Staubli VAL3: listupdate.pgx

public program listupdate(num pFirst (dimensions=1))
  local num lI
  local num lLen
  local string lStr
  local string lStr2
  local num lValue
  local num lView
  local num lX
  local num lY
  local num l_nSize
  local bool l_bEmpty
begin
  //
  // insert into the box all the data
  //
  // to prevent a negative value
  if pFirst>=0
    nFirst=pFirst
  else
    nFirst=0
  endIf
  // save the coordinate
  lValue=nBottomY-1
  // check the overFlow
  l_nSize=size(sItems)-1
  if (nFirst+nView>l_nSize)
    // reset the value
    nFirst=nView=0
  endIf
  lI=0
  // check the unKnow poblem
  if l_nSize<lValue
    if nFirst!=0
      nView=nView+nFirst
      nFirst=0
    endIf
  endIf
  do
    lX=nTopX+1
    lY=nBottomY+lI-1
    lY=nTopY+lI+1
    lLen=nBottomX
    if ((lI+nFirst)<size(sItems))
      // print the item
      if (l_nSize>=0)
        lStr=mid(sItems[(lI+nFirst)],lLen,0)
      endIf
    else
      // print the blank line
      lStr="                                        "
    endIf
    // fill the line
    call strfill(lStr,lLen,lStr2)
    gotoxy(lX,lY)
    put(lStr2)
    lI=lI+1
  until (lI>lValue)
  // underlien the actual line
  call isListEmpty(l_bEmpty)
  if !l_bEmpty
    call listcursor(nView,true)
  else
    call listcursor(nView,false)
    nView=0
    nFirst=0
  endIf
  // print the scroll
  call printScroll()
  // leave the resourse
  delay(0)
end
